Fanuc KAREL source: ka00143.KL

-- PROVISIONAL review KL for V1013-1; original PC SHA256 44d014e494de60b61ed381d5c7c9fed56ff7e86bf9db8bac44c7dd88cb8a116a
-- Incomplete behavior may be omitted. Consult companion uncertainty JSON. Do not deploy.
PROGRAM KA00143
%NOLOCKGROUP
-- UNRESOLVED_DECL SRC type=002017
-- UNRESOLVED_DECL DST type=002018
BEGIN
  -- UNRESOLVED_PC offsets 5-19; opcodes 2E,22,9D,33,B4
  -- UNRESOLVED_PC offsets 24-42; opcodes 22,9D,33,B3,22,9D,33,B2
  -- UNRESOLVED_PC offsets 47-51; opcodes 7F
END KA00143
